{attribute 'qualified_only'}
VAR_GLOBAL
		EtherCAT_Master_EPPxxxx : EtherCAT_Master_EPPxxxx_9A8F5D7B;
END_VAR

(* stored: Version 1.2.0.0, ProductVersion 3.1.4024.11
   GVL GVL_iXlinker: Id {3092b493-34f9-4b0d-ad36-3fa6eb2fdb04} *)
